			END_IF	
			eCameraMethodState := CAMERA_METHOD_SEND_COMMAND;
			eCameraState := CAMERA_METHOD_DONE;

		END_IF
END_CASE
END_METHOD

METHOD PROTECTED MS_SetOnline
CASE eCameraMethodState OF
	CAMERA_METHOD_SEND_COMMAND:
		MEMSET(ADR(sSendMessage),0,SIZEOF(sSendMessage));
		sSendMessage := FUN_MergeStrings3('SO', TO_STRING(bSetCameraOnline), '$R$L');
		FUN_StringToTcpBufferData(ADR(sSendMessage),ADR(stSendData));
		
		IF fbTcpClient.MR_AppendToSendBuffer(stSendData) THEN
			eCameraMethodState := CAMERA_METHOD_RECEIVE_RESPONSE;
							
		END_IF

	CAMERA_METHOD_RECEIVE_RESPONSE:
		stReciveData := fbTcpClient.NextRecivedMessage;
		
		IF stReciveData.iLength > 0 THEN
			MEMSET(ADR(sReciveMessage),0,SIZEOF(sReciveMessage));
			FUN_TcpBufferDataToString(ADR(sReciveMessage),ADR(stReciveData));
			MEMCPY(ADR(sLastStatusCode),ADR(sReciveMessage),2);
			iLastStatusCode := STRING_TO_INT(sLastStatusCode);
			
			IF iLastStatusCode = 1 THEN 
				eCameraSetOnlineStatus := 1;
				
			ELSIF iLastStatusCode = 0 THEN
				eCameraSetOnlineStatus := 0;
				
			ELSIF iLastStatusCode = -1 THEN
				eCameraSetOnlineStatus := -1;
				
			ELSIF iLastStatusCode = -2 THEN
				eCameraSetOnlineStatus := -2;
				
			ELSIF iLastStatusCode = -5 THEN
				eCameraSetOnlineStatus := -5;
				
			ELSIF iLastStatusCode = -6 THEN
				eCameraSetOnlineStatus := -6;
				
			END_IF	
			eCameraMethodState := CAMERA_METHOD_SEND_COMMAND;
			eCameraState := CAMERA_METHOD_DONE;

		END_IF
END_CASE
END_METHOD

METHOD PROTECTED MS_StoreFile
CASE eCameraMethodState OF
	CAMERA_METHOD_SEND_COMMAND:
		MEMSET(ADR(sSendMessage),0,SIZEOF(sSendMessage));
		sSendMessage := FUN_MergeStrings3('TF', sStoreFileName,'$R$L');
		FUN_StringToTcpBufferData(ADR(sSendMessage),ADR(stSendData));
		
		IF fbTcpClient.MR_AppendToSendBuffer(stSendData) THEN
			eCameraMethodState := CAMERA_METHOD_RECEIVE_RESPONSE;
							
		END_IF

	CAMERA_METHOD_RECEIVE_RESPONSE:
		stReciveData := fbTcpClient.NextRecivedMessage;
		
		IF stReciveData.iLength > 0 THEN
			MEMSET(ADR(sReciveMessage),0,SIZEOF(sReciveMessage));
			FUN_TcpBufferDataToString(ADR(sReciveMessage),ADR(stReciveData));
			MEMCPY(ADR(sLastStatusCode),ADR(sReciveMessage),2);
			iLastStatusCode := STRING_TO_INT(sLastStatusCode);
			
			IF iLastStatusCode = 1 THEN 
				eCameraStoreFileStatus := 1;
			ELSIF iLastStatusCode = 0 THEN
				eCameraStoreFileStatus := 0;
			ELSIF iLastStatusCode = -1 THEN
				eCameraStoreFileStatus := -1;
			ELSIF iLastStatusCode = -2 THEN
				eCameraStoreFileStatus := -2;
			ELSIF iLastStatusCode = -6 THEN
				eCameraStoreFileStatus := -6;
			END_IF	
			eCameraMethodState := CAMERA_METHOD_SEND_COMMAND;
			eCameraState := CAMERA_METHOD_DONE;

		END_IF
END_CASE
END_METHOD

METHOD PROTECTED MS_Uninitialized
;
END_METHOD

PROPERTY Name : STRING
GET
Name := sName;
END_GET
SET
sName := Name;
END_SET
END_PROPERTY

PROPERTY ref_TcpClient : REFERENCE TO FB_TcpClient
GET
ref_TcpClient REF= fbTcpClient;
END_GET
END_PROPERTY

METHOD PROTECTED StateMachine
CASE eCameraState OF
	CAMERA_UNINITIALIZED:
		MS_Uninitialized();
		
	CAMERA_INITIALIZING:
		MS_Initializing();
		
	CAMERA_READY:
		MS_Ready();
	
	CAMERA_IDLE:
		MS_Idle();	
		
	CAMERA_RESET:
		MS_Reset();
		
	CAMERA_LOAD_FILE:
		MS_LoadFile();	
		
	CAMERA_GET_FILE:
		MS_GetFile();

	CAMERA_GET_VALUE_EASY_BUILDER:
		MS_GetValueEasyBuilder();	
		
	CAMERA_GET_VALUE_SPREADSHEET:
		MS_GetValueSpreadsheet();	
		
	CAMERA_SET_ONLINE:
		MS_SetOnline();	
	
	CAMERA_GET_ONLINE:
		MS_GetOnline();
		
	CAMERA_RESET_SYSTEM:
		MS_ResetSystem();
	
	CAMERA_GET_CONNECTIONS:
		MS_GetConnections();
		
	CAMERA_GET_EXPR:
		MS_GetExpr();
	
	CAMERA_GET_FILE_LIST:
		MS_GetFileList();
	
	CAMERA_PUT_LIVE:
		MS_PutLive();
	
	CAMERA_PUT_PORTNUM:
		MS_PutPortnum();
	
	CAMERA_PUT_TIMEOUT:
		MS_PutTimeout();
	
	CAMERA_PUT_UPDATE:
		MS_PutUpdate();
	
	CAMERA_PUT_WATCH:
		MS_PutWatch();	
	
	CAMERA_SET_JOB:
		MS_SetJob();
		
	CAMERA_GET_JOB:
		MS_GetJob();
	
	CAMERA_STORE_FILE:
		MS_StoreFile();	
		
	CAMERA_GET_POSITION:
		MS_GetPosition();
	
	CAMERA_IMAGE_TRIGGER:
		MS_ImageTrigger();
	
	CAMERA_GET_VALUES:
		MS_GetValues();
	
	CAMERA_METHOD_DONE:
		MS_MethodDone();
	
	CAMERA_ABORTING:
		MS_Aborting();
	
END_CASE
END_METHOD

END_FUNCTION_BLOCK
